Universal Robots URScript: test_script.urscript

# HEADER_BEGIN

def test_func():
  textmsg("test function")
end

# HEADER_END

# NODE_CONTROL_LOOP_BEGINS

test_func()

# NODE_CONTROL_LOOP_ENDS
